Fanuc KAREL source: kx00007.KL

-- PROVISIONAL review KL for V1013-1; original PC SHA256 563670a1b23899aed7b46bfce0e5bc1c966f222f0e0ad8c88de38337668b1bdf
-- Incomplete behavior may be omitted. Consult companion uncertainty JSON. Do not deploy.
PROGRAM KX00007
%NOLOCKGROUP
VAR
  I : INTEGER
  J : INTEGER
  B : BOOLEAN
  F : FILE
  S : STRING[80]
-- UNRESOLVED_DECL P type=000102
BEGIN
  -- UNRESOLVED_PC offsets 5-13; opcodes 9D,2E,1F
  -- UNRESOLVED_PC offsets 18-22; opcodes 7F
END KX00007
